(* PLC project logical_and, Dassault Systèmes ControlBuild 2024x *)
(* stored: creationDateTime 2023-10-03T11:13:29-01:00 *)

(* This module makes a "logical AND" operation between two inputs. Result is a boolean. *)
FUNCTION_BLOCK equipment_library.logical_and
  VAR_INPUT
    inputBit1 : BOOL := false;
    inputBit2 : BOOL := false;
  END_VAR
  VAR_OUTPUT
    ouputBit : BOOL := false;
  END_VAR
  VAR CONSTANT
    input1Logic : BOOL := true;
    input2Logic : BOOL := true;
    outputLogic : BOOL := true;
  END_VAR
  VAR
    d_output : BOOL := false;
    v_d_output : BOOL := true;
  END_VAR


ACTION C_source_code:
/* ----------------------------------------------------------------	*/
/* Type : Model of Operative Behaviour					*/
/* Category :  Toolbox							*/
/* Author : Dassault Systemes						*/
/* Update date : June 2018						*/
/* ----------------------------------------------------------------	*/
/* This module makes a "logical AND" operation between two inputs.	*/
/* Result is a boolean.							*/
/* The output can be preset	by the user					*/
/* ----------------------------------------------------------------	*/

if (d_output) ouputBit = v_d_output;
else
	ouputBit = ((inputBit1 ^ ! input1Logic) & (inputBit2 ^ ! input2Logic)) ^ ! outputLogic;
END_ACTION
END_FUNCTION_BLOCK
